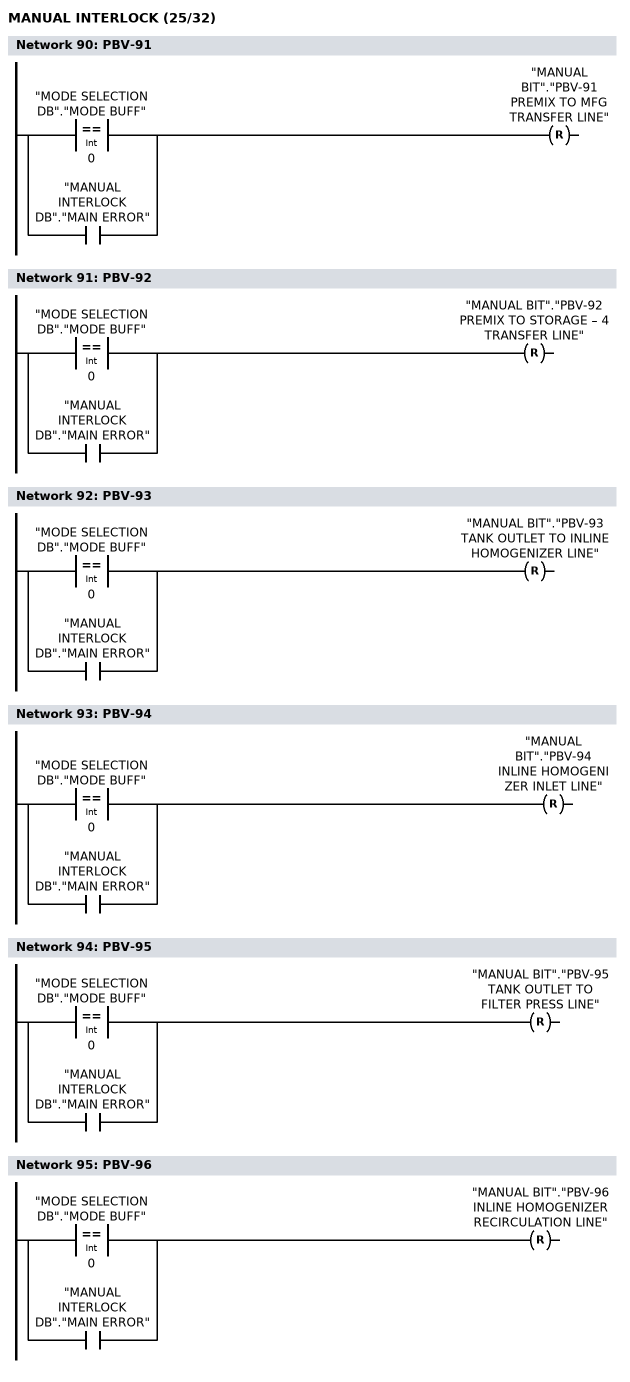
   RUNG wire#powerrail
      { S7_Templates := "SrcType := Int" } EQ_Contact(in1 := "MODE SELECTION DB"."MODE BUFF", in2 := 0)
      wire#w1
      R_Coil( "MANUAL BIT"."PBV-91 PREMIX TO MFG TRANSFER LINE" )
   END_RUNG
   RUNG wire#powerrail
      Contact( "MANUAL INTERLOCK DB"."MAIN ERROR" )
   END_RUNG wire#w1
   // the same network as SCL:
   IF ("MODE SELECTION DB"."MODE BUFF" = 0) OR "MANUAL INTERLOCK DB"."MAIN ERROR" THEN
       "MANUAL BIT"."PBV-91 PREMIX TO MFG TRANSFER LINE" := FALSE;
   END_IF;
END_REGION

REGION Network 91: PBV-92
   RUNG wire#powerrail
      { S7_Templates := "SrcType := Int" } EQ_Contact(in1 := "MODE SELECTION DB"."MODE BUFF", in2 := 0)
      wire#w1
      R_Coil( "MANUAL BIT"."PBV-92 PREMIX TO STORAGE – 4 TRANSFER LINE" )
   END_RUNG
   RUNG wire#powerrail
      Contact( "MANUAL INTERLOCK DB"."MAIN ERROR" )
   END_RUNG wire#w1
   // the same network as SCL:
   IF ("MODE SELECTION DB"."MODE BUFF" = 0) OR "MANUAL INTERLOCK DB"."MAIN ERROR" THEN
       "MANUAL BIT"."PBV-92 PREMIX TO STORAGE – 4 TRANSFER LINE" := FALSE;
   END_IF;
END_REGION

REGION Network 92: PBV-93
   RUNG wire#powerrail
      { S7_Templates := "SrcType := Int" } EQ_Contact(in1 := "MODE SELECTION DB"."MODE BUFF", in2 := 0)
      wire#w1
      R_Coil( "MANUAL BIT"."PBV-93 TANK OUTLET TO INLINE HOMOGENIZER LINE" )
   END_RUNG
   RUNG wire#powerrail
      Contact( "MANUAL INTERLOCK DB"."MAIN ERROR" )
   END_RUNG wire#w1
   // the same network as SCL:
   IF ("MODE SELECTION DB"."MODE BUFF" = 0) OR "MANUAL INTERLOCK DB"."MAIN ERROR" THEN
       "MANUAL BIT"."PBV-93 TANK OUTLET TO INLINE HOMOGENIZER LINE" := FALSE;
   END_IF;
END_REGION

REGION Network 93: PBV-94
   RUNG wire#powerrail
      { S7_Templates := "SrcType := Int" } EQ_Contact(in1 := "MODE SELECTION DB"."MODE BUFF", in2 := 0)
      wire#w1
      R_Coil( "MANUAL BIT"."PBV-94 INLINE HOMOGENIZER INLET LINE" )
   END_RUNG
   RUNG wire#powerrail
      Contact( "MANUAL INTERLOCK DB"."MAIN ERROR" )
   END_RUNG wire#w1
   // the same network as SCL:
   IF ("MODE SELECTION DB"."MODE BUFF" = 0) OR "MANUAL INTERLOCK DB"."MAIN ERROR" THEN
       "MANUAL BIT"."PBV-94 INLINE HOMOGENIZER INLET LINE" := FALSE;
   END_IF;
END_REGION

REGION Network 94: PBV-95
   RUNG wire#powerrail
      { S7_Templates := "SrcType := Int" } EQ_Contact(in1 := "MODE SELECTION DB"."MODE BUFF", in2 := 0)
      wire#w1
      R_Coil( "MANUAL BIT"."PBV-95 TANK OUTLET TO FILTER PRESS LINE" )
   END_RUNG
   RUNG wire#powerrail
      Contact( "MANUAL INTERLOCK DB"."MAIN ERROR" )
   END_RUNG wire#w1
   // the same network as SCL:
   IF ("MODE SELECTION DB"."MODE BUFF" = 0) OR "MANUAL INTERLOCK DB"."MAIN ERROR" THEN
       "MANUAL BIT"."PBV-95 TANK OUTLET TO FILTER PRESS LINE" := FALSE;
   END_IF;
END_REGION

REGION Network 95: PBV-96
   RUNG wire#powerrail
      { S7_Templates := "SrcType := Int" } EQ_Contact(in1 := "MODE SELECTION DB"."MODE BUFF", in2 := 0)
      wire#w1
      R_Coil( "MANUAL BIT"."PBV-96 INLINE HOMOGENIZER RECIRCULATION LINE" )
   END_RUNG
   RUNG wire#powerrail
      Contact( "MANUAL INTERLOCK DB"."MAIN ERROR" )
   END_RUNG wire#w1
   // the same network as SCL:
   IF ("MODE SELECTION DB"."MODE BUFF" = 0) OR "MANUAL INTERLOCK DB"."MAIN ERROR" THEN
       "MANUAL BIT"."PBV-96 INLINE HOMOGENIZER RECIRCULATION LINE" := FALSE;
   END_IF;
END_REGION

REGION Network 96: PBV-97
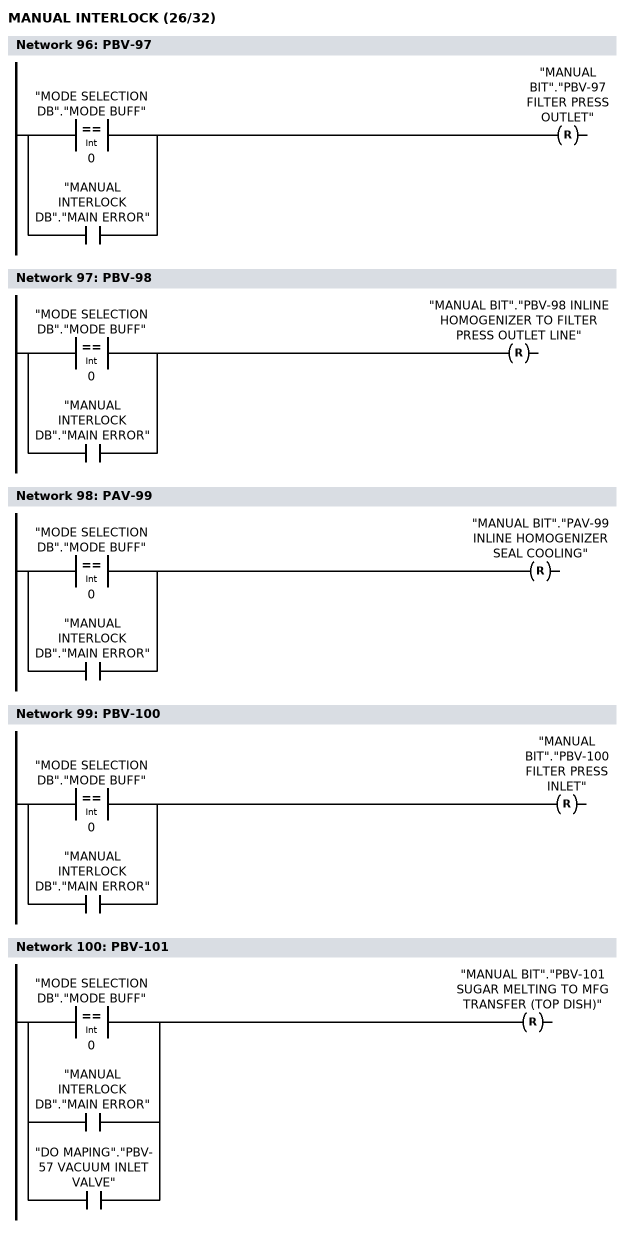
   RUNG wire#powerrail
      { S7_Templates := "SrcType := Int" } EQ_Contact(in1 := "MODE SELECTION DB"."MODE BUFF", in2 := 0)
      wire#w1
      R_Coil( "MANUAL BIT"."PBV-97 FILTER PRESS OUTLET" )
   END_RUNG
   RUNG wire#powerrail
      Contact( "MANUAL INTERLOCK DB"."MAIN ERROR" )
   END_RUNG wire#w1
   // the same network as SCL:
   IF ("MODE SELECTION DB"."MODE BUFF" = 0) OR "MANUAL INTERLOCK DB"."MAIN ERROR" THEN
       "MANUAL BIT"."PBV-97 FILTER PRESS OUTLET" := FALSE;
   END_IF;
END_REGION

REGION Network 97: PBV-98
   RUNG wire#powerrail
      { S7_Templates := "SrcType := Int" } EQ_Contact(in1 := "MODE SELECTION DB"."MODE BUFF", in2 := 0)
      wire#w1
      R_Coil( "MANUAL BIT"."PBV-98 INLINE HOMOGENIZER TO FILTER PRESS OUTLET LINE" )
   END_RUNG
   RUNG wire#powerrail
      Contact( "MANUAL INTERLOCK DB"."MAIN ERROR" )
   END_RUNG wire#w1
   // the same network as SCL:
   IF ("MODE SELECTION DB"."MODE BUFF" = 0) OR "MANUAL INTERLOCK DB"."MAIN ERROR" THEN
       "MANUAL BIT"."PBV-98 INLINE HOMOGENIZER TO FILTER PRESS OUTLET LINE" := FALSE;
   END_IF;
END_REGION

REGION Network 98: PAV-99
   RUNG wire#powerrail
      { S7_Templates := "SrcType := Int" } EQ_Contact(in1 := "MODE SELECTION DB"."MODE BUFF", in2 := 0)
      wire#w1
      R_Coil( "MANUAL BIT"."PAV-99 INLINE HOMOGENIZER SEAL COOLING" )
   END_RUNG
   RUNG wire#powerrail
      Contact( "MANUAL INTERLOCK DB"."MAIN ERROR" )
   END_RUNG wire#w1
   // the same network as SCL:
   IF ("MODE SELECTION DB"."MODE BUFF" = 0) OR "MANUAL INTERLOCK DB"."MAIN ERROR" THEN
       "MANUAL BIT"."PAV-99 INLINE HOMOGENIZER SEAL COOLING" := FALSE;
   END_IF;
END_REGION

REGION Network 99: PBV-100
   RUNG wire#powerrail
      { S7_Templates := "SrcType := Int" } EQ_Contact(in1 := "MODE SELECTION DB"."MODE BUFF", in2 := 0)
      wire#w1
      R_Coil( "MANUAL BIT"."PBV-100 FILTER PRESS INLET" )
   END_RUNG
   RUNG wire#powerrail
      Contact( "MANUAL INTERLOCK DB"."MAIN ERROR" )
   END_RUNG wire#w1
   // the same network as SCL:
   IF ("MODE SELECTION DB"."MODE BUFF" = 0) OR "MANUAL INTERLOCK DB"."MAIN ERROR" THEN
       "MANUAL BIT"."PBV-100 FILTER PRESS INLET" := FALSE;
   END_IF;
END_REGION

REGION Network 100: PBV-101
   RUNG wire#powerrail
      { S7_Templates := "SrcType := Int" } EQ_Contact(in1 := "MODE SELECTION DB"."MODE BUFF", in2 := 0)
      wire#w1
      R_Coil( "MANUAL BIT"."PBV-101 SUGAR MELTING TO MFG TRANSFER (TOP DISH)" )
   END_RUNG
   RUNG wire#powerrail
      Contact( "MANUAL INTERLOCK DB"."MAIN ERROR" )
   END_RUNG wire#w1
   RUNG wire#powerrail
      Contact( "DO MAPING"."PBV-57 VACUUM INLET VALVE" )
   END_RUNG wire#w1
   // the same network as SCL:
   IF ("MODE SELECTION DB"."MODE BUFF" = 0) OR "MANUAL INTERLOCK DB"."MAIN ERROR" OR "DO MAPING"."PBV-57 VACUUM INLET VALVE" THEN
       "MANUAL BIT"."PBV-101 SUGAR MELTING TO MFG TRANSFER (TOP DISH)" := FALSE;
   END_IF;
END_REGION

REGION Network 101: PBV-102
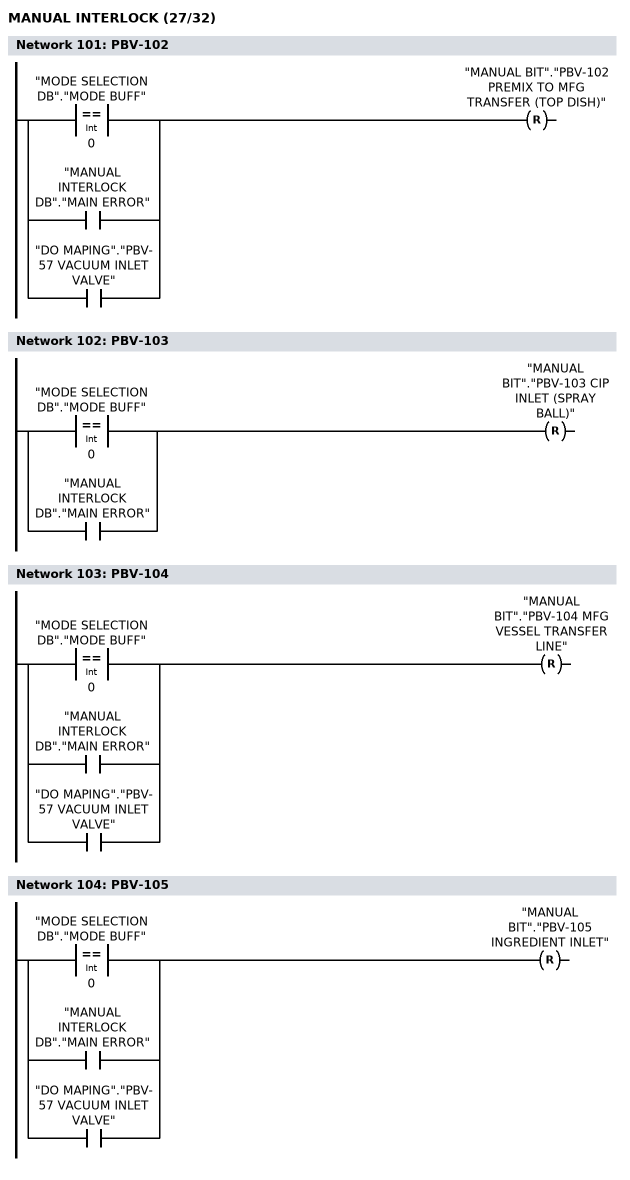
   RUNG wire#powerrail
      { S7_Templates := "SrcType := Int" } EQ_Contact(in1 := "MODE SELECTION DB"."MODE BUFF", in2 := 0)
      wire#w1
      R_Coil( "MANUAL BIT"."PBV-102 PREMIX TO MFG TRANSFER (TOP DISH)" )
   END_RUNG
   RUNG wire#powerrail
      Contact( "MANUAL INTERLOCK DB"."MAIN ERROR" )
   END_RUNG wire#w1
   RUNG wire#powerrail
      Contact( "DO MAPING"."PBV-57 VACUUM INLET VALVE" )
   END_RUNG wire#w1
   // the same network as SCL:
   IF ("MODE SELECTION DB"."MODE BUFF" = 0) OR "MANUAL INTERLOCK DB"."MAIN ERROR" OR "DO MAPING"."PBV-57 VACUUM INLET VALVE" THEN
       "MANUAL BIT"."PBV-102 PREMIX TO MFG TRANSFER (TOP DISH)" := FALSE;
   END_IF;
END_REGION

REGION Network 102: PBV-103
   RUNG wire#powerrail
      { S7_Templates := "SrcType := Int" } EQ_Contact(in1 := "MODE SELECTION DB"."MODE BUFF", in2 := 0)
      wire#w1
      R_Coil( "MANUAL BIT"."PBV-103 CIP INLET (SPRAY BALL)" )
   END_RUNG
   RUNG wire#powerrail
      Contact( "MANUAL INTERLOCK DB"."MAIN ERROR" )
   END_RUNG wire#w1
   // the same network as SCL:
   IF ("MODE SELECTION DB"."MODE BUFF" = 0) OR "MANUAL INTERLOCK DB"."MAIN ERROR" THEN
       "MANUAL BIT"."PBV-103 CIP INLET (SPRAY BALL)" := FALSE;
   END_IF;
END_REGION

REGION Network 103: PBV-104
   RUNG wire#powerrail
      { S7_Templates := "SrcType := Int" } EQ_Contact(in1 := "MODE SELECTION DB"."MODE BUFF", in2 := 0)
      wire#w1
      R_Coil( "MANUAL BIT"."PBV-104 MFG VESSEL TRANSFER LINE" )
   END_RUNG
   RUNG wire#powerrail
      Contact( "MANUAL INTERLOCK DB"."MAIN ERROR" )
   END_RUNG wire#w1
   RUNG wire#powerrail
      Contact( "DO MAPING"."PBV-57 VACUUM INLET VALVE" )
   END_RUNG wire#w1
   // the same network as SCL:
   IF ("MODE SELECTION DB"."MODE BUFF" = 0) OR "MANUAL INTERLOCK DB"."MAIN ERROR" OR "DO MAPING"."PBV-57 VACUUM INLET VALVE" THEN
       "MANUAL BIT"."PBV-104 MFG VESSEL TRANSFER LINE" := FALSE;
   END_IF;
END_REGION

REGION Network 104: PBV-105
   RUNG wire#powerrail
      { S7_Templates := "SrcType := Int" } EQ_Contact(in1 := "MODE SELECTION DB"."MODE BUFF", in2 := 0)
      wire#w1
      R_Coil( "MANUAL BIT"."PBV-105 INGREDIENT INLET" )
   END_RUNG
   RUNG wire#powerrail
      Contact( "MANUAL INTERLOCK DB"."MAIN ERROR" )
   END_RUNG wire#w1
   RUNG wire#powerrail
      Contact( "DO MAPING"."PBV-57 VACUUM INLET VALVE" )
   END_RUNG wire#w1
   // the same network as SCL:
   IF ("MODE SELECTION DB"."MODE BUFF" = 0) OR "MANUAL INTERLOCK DB"."MAIN ERROR" OR "DO MAPING"."PBV-57 VACUUM INLET VALVE" THEN
       "MANUAL BIT"."PBV-105 INGREDIENT INLET" := FALSE;
   END_IF;
END_REGION

REGION Network 105: PBV-106
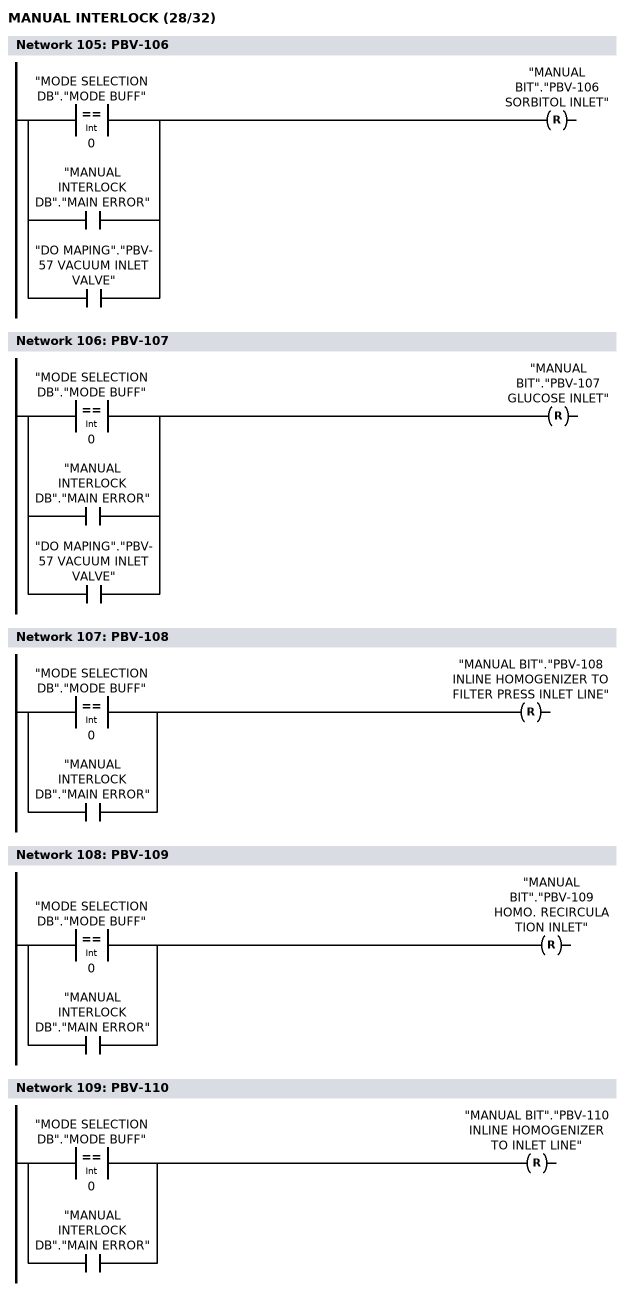
   RUNG wire#powerrail
      { S7_Templates := "SrcType := Int" } EQ_Contact(in1 := "MODE SELECTION DB"."MODE BUFF", in2 := 0)
      wire#w1
      R_Coil( "MANUAL BIT"."PBV-106 SORBITOL INLET" )
   END_RUNG
   RUNG wire#powerrail
      Contact( "MANUAL INTERLOCK DB"."MAIN ERROR" )
   END_RUNG wire#w1
   RUNG wire#powerrail
      Contact( "DO MAPING"."PBV-57 VACUUM INLET VALVE" )
   END_RUNG wire#w1
   // the same network as SCL:
   IF ("MODE SELECTION DB"."MODE BUFF" = 0) OR "MANUAL INTERLOCK DB"."MAIN ERROR" OR "DO MAPING"."PBV-57 VACUUM INLET VALVE" THEN
       "MANUAL BIT"."PBV-106 SORBITOL INLET" := FALSE;
   END_IF;
END_REGION

REGION Network 106: PBV-107
   RUNG wire#powerrail
      { S7_Templates := "SrcType := Int" } EQ_Contact(in1 := "MODE SELECTION DB"."MODE BUFF", in2 := 0)
      wire#w1
      R_Coil( "MANUAL BIT"."PBV-107 GLUCOSE INLET" )
   END_RUNG
   RUNG wire#powerrail
      Contact( "MANUAL INTERLOCK DB"."MAIN ERROR" )
   END_RUNG wire#w1
   RUNG wire#powerrail
      Contact( "DO MAPING"."PBV-57 VACUUM INLET VALVE" )
   END_RUNG wire#w1
   // the same network as SCL:
   IF ("MODE SELECTION DB"."MODE BUFF" = 0) OR "MANUAL INTERLOCK DB"."MAIN ERROR" OR "DO MAPING"."PBV-57 VACUUM INLET VALVE" THEN
       "MANUAL BIT"."PBV-107 GLUCOSE INLET" := FALSE;
   END_IF;
END_REGION

REGION Network 107: PBV-108
   RUNG wire#powerrail
      { S7_Templates := "SrcType := Int" } EQ_Contact(in1 := "MODE SELECTION DB"."MODE BUFF", in2 := 0)
      wire#w1
      R_Coil( "MANUAL BIT"."PBV-108 INLINE HOMOGENIZER TO FILTER PRESS INLET LINE" )
   END_RUNG
   RUNG wire#powerrail
      Contact( "MANUAL INTERLOCK DB"."MAIN ERROR" )
   END_RUNG wire#w1
   // the same network as SCL:
   IF ("MODE SELECTION DB"."MODE BUFF" = 0) OR "MANUAL INTERLOCK DB"."MAIN ERROR" THEN
       "MANUAL BIT"."PBV-108 INLINE HOMOGENIZER TO FILTER PRESS INLET LINE" := FALSE;
   END_IF;
END_REGION

REGION Network 108: PBV-109
   RUNG wire#powerrail
      { S7_Templates := "SrcType := Int" } EQ_Contact(in1 := "MODE SELECTION DB"."MODE BUFF", in2 := 0)
      wire#w1
      R_Coil( "MANUAL BIT"."PBV-109 HOMO. RECIRCULATION INLET" )
   END_RUNG
   RUNG wire#powerrail
      Contact( "MANUAL INTERLOCK DB"."MAIN ERROR" )
   END_RUNG wire#w1
   // the same network as SCL:
   IF ("MODE SELECTION DB"."MODE BUFF" = 0) OR "MANUAL INTERLOCK DB"."MAIN ERROR" THEN
       "MANUAL BIT"."PBV-109 HOMO. RECIRCULATION INLET" := FALSE;
   END_IF;
END_REGION

REGION Network 109: PBV-110
   RUNG wire#powerrail
      { S7_Templates := "SrcType := Int" } EQ_Contact(in1 := "MODE SELECTION DB"."MODE BUFF", in2 := 0)
      wire#w1
      R_Coil( "MANUAL BIT"."PBV-110 INLINE HOMOGENIZER TO INLET LINE" )
   END_RUNG
   RUNG wire#powerrail
      Contact( "MANUAL INTERLOCK DB"."MAIN ERROR" )
   END_RUNG wire#w1
   // the same network as SCL:
   IF ("MODE SELECTION DB"."MODE BUFF" = 0) OR "MANUAL INTERLOCK DB"."MAIN ERROR" THEN
       "MANUAL BIT"."PBV-110 INLINE HOMOGENIZER TO INLET LINE" := FALSE;
   END_IF;
END_REGION

REGION Network 110: PBV-111
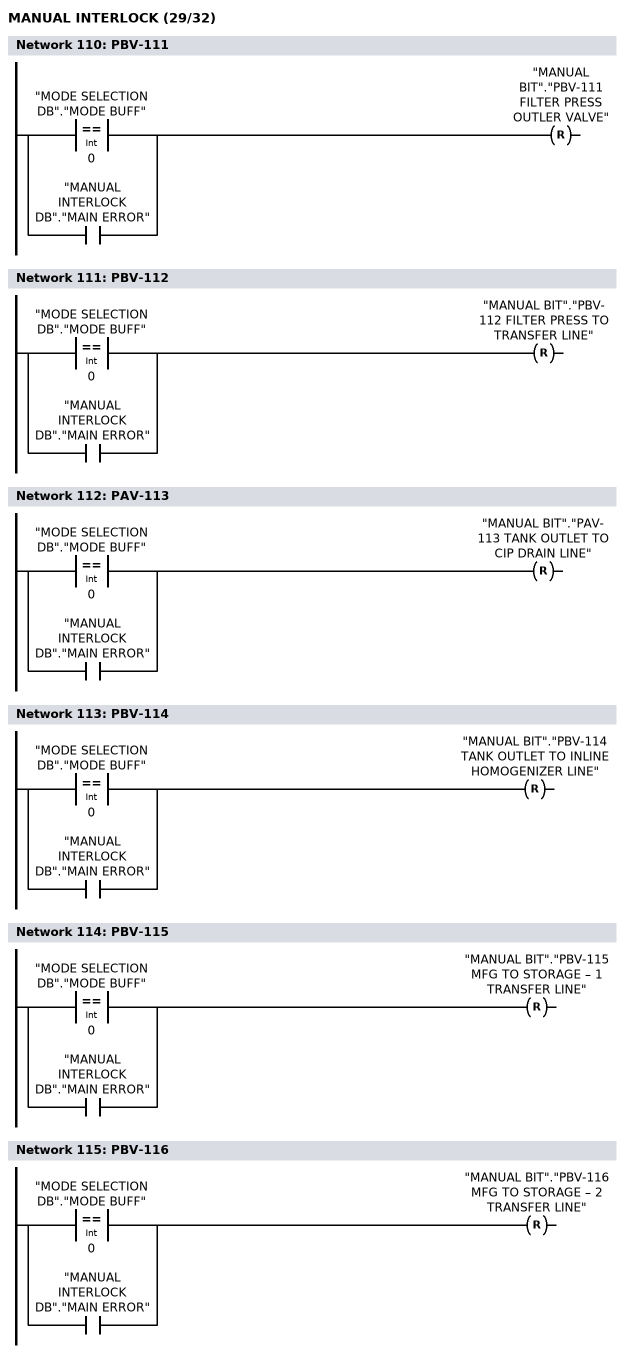
   RUNG wire#powerrail
      { S7_Templates := "SrcType := Int" } EQ_Contact(in1 := "MODE SELECTION DB"."MODE BUFF", in2 := 0)
      wire#w1
      R_Coil( "MANUAL BIT"."PBV-111 FILTER PRESS OUTLER VALVE" )
   END_RUNG
   RUNG wire#powerrail
      Contact( "MANUAL INTERLOCK DB"."MAIN ERROR" )
   END_RUNG wire#w1
   // the same network as SCL:
   IF ("MODE SELECTION DB"."MODE BUFF" = 0) OR "MANUAL INTERLOCK DB"."MAIN ERROR" THEN
       "MANUAL BIT"."PBV-111 FILTER PRESS OUTLER VALVE" := FALSE;
   END_IF;
END_REGION

REGION Network 111: PBV-112
   RUNG wire#powerrail
      { S7_Templates := "SrcType := Int" } EQ_Contact(in1 := "MODE SELECTION DB"."MODE BUFF", in2 := 0)
      wire#w1
      R_Coil( "MANUAL BIT"."PBV-112 FILTER PRESS TO TRANSFER LINE" )
   END_RUNG
   RUNG wire#powerrail
      Contact( "MANUAL INTERLOCK DB"."MAIN ERROR" )
   END_RUNG wire#w1
   // the same network as SCL:
   IF ("MODE SELECTION DB"."MODE BUFF" = 0) OR "MANUAL INTERLOCK DB"."MAIN ERROR" THEN
       "MANUAL BIT"."PBV-112 FILTER PRESS TO TRANSFER LINE" := FALSE;
   END_IF;
END_REGION

REGION Network 112: PAV-113
   RUNG wire#powerrail
      { S7_Templates := "SrcType := Int" } EQ_Contact(in1 := "MODE SELECTION DB"."MODE BUFF", in2 := 0)
      wire#w1
      R_Coil( "MANUAL BIT"."PAV-113 TANK OUTLET TO CIP DRAIN LINE" )
   END_RUNG
   RUNG wire#powerrail
      Contact( "MANUAL INTERLOCK DB"."MAIN ERROR" )
   END_RUNG wire#w1
   // the same network as SCL:
   IF ("MODE SELECTION DB"."MODE BUFF" = 0) OR "MANUAL INTERLOCK DB"."MAIN ERROR" THEN
       "MANUAL BIT"."PAV-113 TANK OUTLET TO CIP DRAIN LINE" := FALSE;
   END_IF;
END_REGION

REGION Network 113: PBV-114
   RUNG wire#powerrail
      { S7_Templates := "SrcType := Int" } EQ_Contact(in1 := "MODE SELECTION DB"."MODE BUFF", in2 := 0)
      wire#w1
      R_Coil( "MANUAL BIT"."PBV-114 TANK OUTLET TO INLINE HOMOGENIZER LINE" )
   END_RUNG
   RUNG wire#powerrail
      Contact( "MANUAL INTERLOCK DB"."MAIN ERROR" )
   END_RUNG wire#w1
   // the same network as SCL:
   IF ("MODE SELECTION DB"."MODE BUFF" = 0) OR "MANUAL INTERLOCK DB"."MAIN ERROR" THEN
       "MANUAL BIT"."PBV-114 TANK OUTLET TO INLINE HOMOGENIZER LINE" := FALSE;
   END_IF;
END_REGION

REGION Network 114: PBV-115
   RUNG wire#powerrail
      { S7_Templates := "SrcType := Int" } EQ_Contact(in1 := "MODE SELECTION DB"."MODE BUFF", in2 := 0)
      wire#w1
      R_Coil( "MANUAL BIT"."PBV-115 MFG TO STORAGE – 1 TRANSFER LINE" )
   END_RUNG
   RUNG wire#powerrail
      Contact( "MANUAL INTERLOCK DB"."MAIN ERROR" )
   END_RUNG wire#w1
   // the same network as SCL:
   IF ("MODE SELECTION DB"."MODE BUFF" = 0) OR "MANUAL INTERLOCK DB"."MAIN ERROR" THEN
       "MANUAL BIT"."PBV-115 MFG TO STORAGE – 1 TRANSFER LINE" := FALSE;
   END_IF;
END_REGION

REGION Network 115: PBV-116
   RUNG wire#powerrail
      { S7_Templates := "SrcType := Int" } EQ_Contact(in1 := "MODE SELECTION DB"."MODE BUFF", in2 := 0)
      wire#w1
      R_Coil( "MANUAL BIT"."PBV-116 MFG TO STORAGE – 2 TRANSFER LINE" )
   END_RUNG
   RUNG wire#powerrail
      Contact( "MANUAL INTERLOCK DB"."MAIN ERROR" )
   END_RUNG wire#w1
   // the same network as SCL:
   IF ("MODE SELECTION DB"."MODE BUFF" = 0) OR "MANUAL INTERLOCK DB"."MAIN ERROR" THEN
       "MANUAL BIT"."PBV-116 MFG TO STORAGE – 2 TRANSFER LINE" := FALSE;
   END_IF;
END_REGION

REGION Network 116: PBV-117
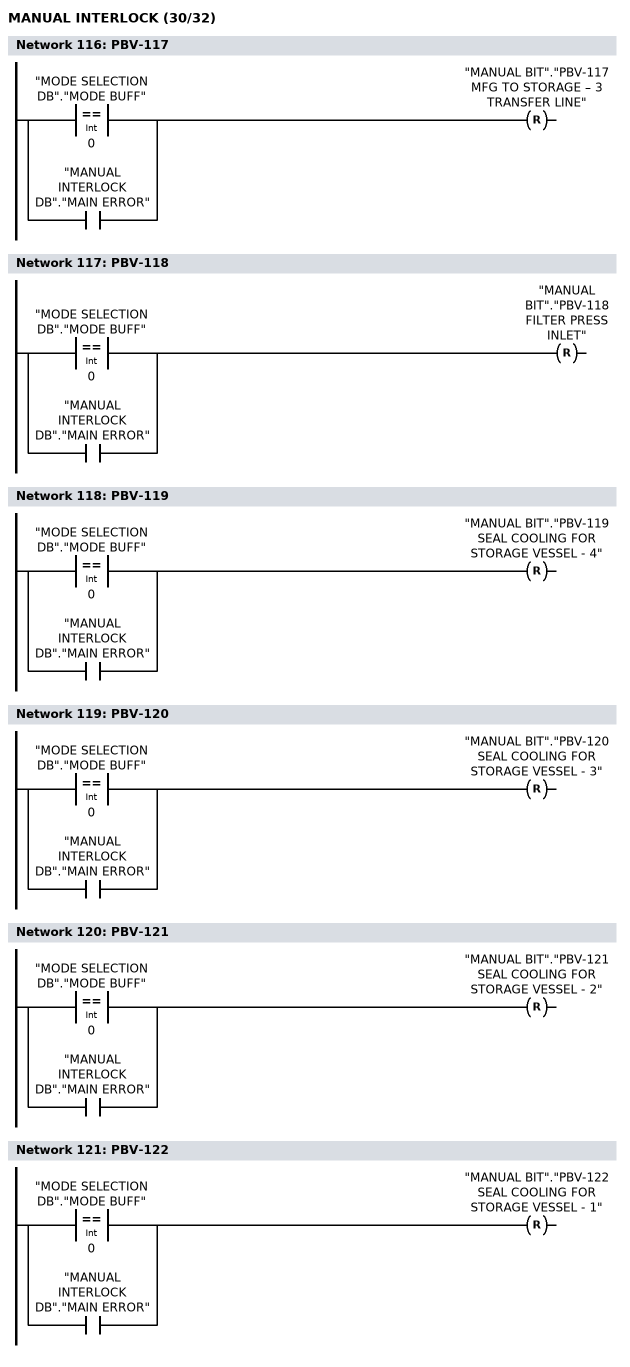
   RUNG wire#powerrail
      { S7_Templates := "SrcType := Int" } EQ_Contact(in1 := "MODE SELECTION DB"."MODE BUFF", in2 := 0)
      wire#w1
      R_Coil( "MANUAL BIT"."PBV-117 MFG TO STORAGE – 3 TRANSFER LINE" )
   END_RUNG
   RUNG wire#powerrail
      Contact( "MANUAL INTERLOCK DB"."MAIN ERROR" )
   END_RUNG wire#w1
   // the same network as SCL:
   IF ("MODE SELECTION DB"."MODE BUFF" = 0) OR "MANUAL INTERLOCK DB"."MAIN ERROR" THEN
       "MANUAL BIT"."PBV-117 MFG TO STORAGE – 3 TRANSFER LINE" := FALSE;
   END_IF;
END_REGION

REGION Network 117: PBV-118
   RUNG wire#powerrail
      { S7_Templates := "SrcType := Int" } EQ_Contact(in1 := "MODE SELECTION DB"."MODE BUFF", in2 := 0)
      wire#w1
      R_Coil( "MANUAL BIT"."PBV-118 FILTER PRESS INLET" )
   END_RUNG
   RUNG wire#powerrail
      Contact( "MANUAL INTERLOCK DB"."MAIN ERROR" )
   END_RUNG wire#w1
   // the same network as SCL:
   IF ("MODE SELECTION DB"."MODE BUFF" = 0) OR "MANUAL INTERLOCK DB"."MAIN ERROR" THEN
       "MANUAL BIT"."PBV-118 FILTER PRESS INLET" := FALSE;
   END_IF;
END_REGION

REGION Network 118: PBV-119
   RUNG wire#powerrail
      { S7_Templates := "SrcType := Int" } EQ_Contact(in1 := "MODE SELECTION DB"."MODE BUFF", in2 := 0)
      wire#w1
      R_Coil( "MANUAL BIT"."PBV-119 SEAL COOLING FOR STORAGE VESSEL - 4" )
   END_RUNG
   RUNG wire#powerrail
      Contact( "MANUAL INTERLOCK DB"."MAIN ERROR" )
   END_RUNG wire#w1
   // the same network as SCL:
   IF ("MODE SELECTION DB"."MODE BUFF" = 0) OR "MANUAL INTERLOCK DB"."MAIN ERROR" THEN
       "MANUAL BIT"."PBV-119 SEAL COOLING FOR STORAGE VESSEL - 4" := FALSE;
   END_IF;
END_REGION

REGION Network 119: PBV-120
   RUNG wire#powerrail
      { S7_Templates := "SrcType := Int" } EQ_Contact(in1 := "MODE SELECTION DB"."MODE BUFF", in2 := 0)
      wire#w1
      R_Coil( "MANUAL BIT"."PBV-120 SEAL COOLING FOR STORAGE VESSEL - 3" )
   END_RUNG
   RUNG wire#powerrail
      Contact( "MANUAL INTERLOCK DB"."MAIN ERROR" )
   END_RUNG wire#w1
   // the same network as SCL:
   IF ("MODE SELECTION DB"."MODE BUFF" = 0) OR "MANUAL INTERLOCK DB"."MAIN ERROR" THEN
       "MANUAL BIT"."PBV-120 SEAL COOLING FOR STORAGE VESSEL - 3" := FALSE;
   END_IF;
END_REGION

REGION Network 120: PBV-121
   RUNG wire#powerrail
      { S7_Templates := "SrcType := Int" } EQ_Contact(in1 := "MODE SELECTION DB"."MODE BUFF", in2 := 0)
      wire#w1
      R_Coil( "MANUAL BIT"."PBV-121 SEAL COOLING FOR STORAGE VESSEL - 2" )
   END_RUNG
   RUNG wire#powerrail
      Contact( "MANUAL INTERLOCK DB"."MAIN ERROR" )
   END_RUNG wire#w1
   // the same network as SCL:
   IF ("MODE SELECTION DB"."MODE BUFF" = 0) OR "MANUAL INTERLOCK DB"."MAIN ERROR" THEN
       "MANUAL BIT"."PBV-121 SEAL COOLING FOR STORAGE VESSEL - 2" := FALSE;
   END_IF;
END_REGION

REGION Network 121: PBV-122
   RUNG wire#powerrail
      { S7_Templates := "SrcType := Int" } EQ_Contact(in1 := "MODE SELECTION DB"."MODE BUFF", in2 := 0)
      wire#w1
      R_Coil( "MANUAL BIT"."PBV-122 SEAL COOLING FOR STORAGE VESSEL - 1" )
   END_RUNG
   RUNG wire#powerrail
      Contact( "MANUAL INTERLOCK DB"."MAIN ERROR" )
   END_RUNG wire#w1
   // the same network as SCL:
   IF ("MODE SELECTION DB"."MODE BUFF" = 0) OR "MANUAL INTERLOCK DB"."MAIN ERROR" THEN
       "MANUAL BIT"."PBV-122 SEAL COOLING FOR STORAGE VESSEL - 1" := FALSE;
   END_IF;
END_REGION

REGION Network 122: PBV-123
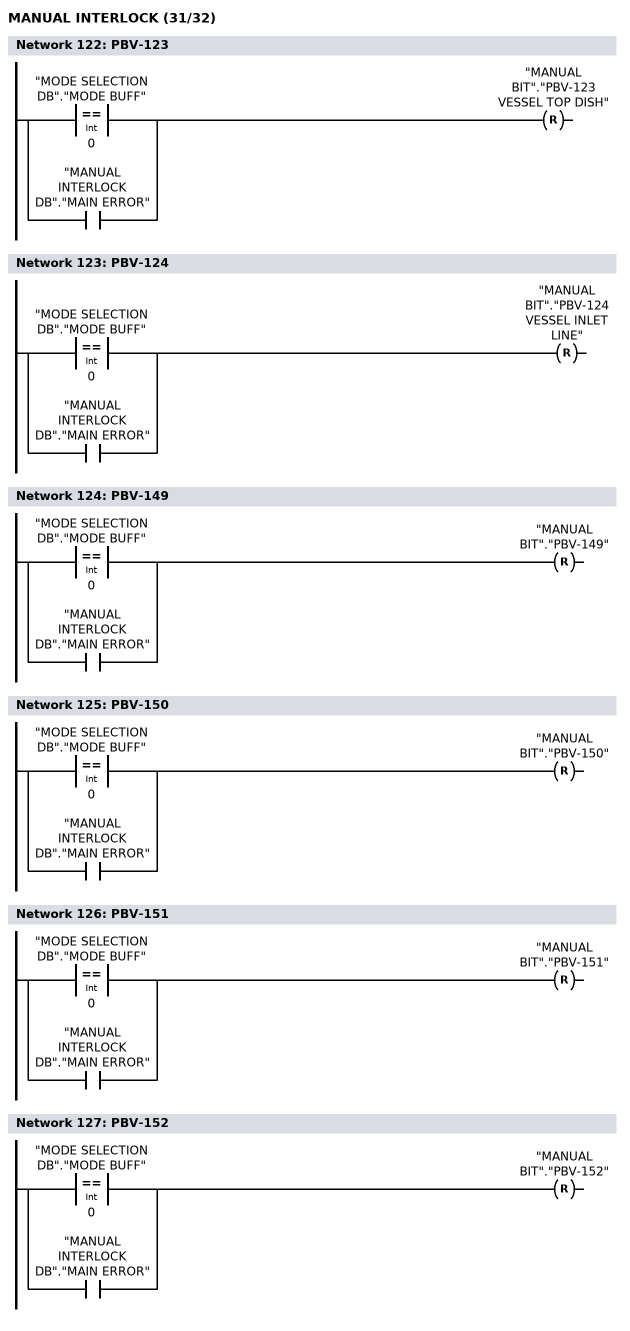
   RUNG wire#powerrail
      { S7_Templates := "SrcType := Int" } EQ_Contact(in1 := "MODE SELECTION DB"."MODE BUFF", in2 := 0)
      wire#w1
      R_Coil( "MANUAL BIT"."PBV-123 VESSEL TOP DISH" )
   END_RUNG
   RUNG wire#powerrail
      Contact( "MANUAL INTERLOCK DB"."MAIN ERROR" )
   END_RUNG wire#w1
   // the same network as SCL:
   IF ("MODE SELECTION DB"."MODE BUFF" = 0) OR "MANUAL INTERLOCK DB"."MAIN ERROR" THEN
       "MANUAL BIT"."PBV-123 VESSEL TOP DISH" := FALSE;
   END_IF;
END_REGION

REGION Network 123: PBV-124
   RUNG wire#powerrail
      { S7_Templates := "SrcType := Int" } EQ_Contact(in1 := "MODE SELECTION DB"."MODE BUFF", in2 := 0)
      wire#w1
      R_Coil( "MANUAL BIT"."PBV-124 VESSEL INLET LINE" )
   END_RUNG
   RUNG wire#powerrail
      Contact( "MANUAL INTERLOCK DB"."MAIN ERROR" )
   END_RUNG wire#w1
   // the same network as SCL:
   IF ("MODE SELECTION DB"."MODE BUFF" = 0) OR "MANUAL INTERLOCK DB"."MAIN ERROR" THEN
       "MANUAL BIT"."PBV-124 VESSEL INLET LINE" := FALSE;
   END_IF;
END_REGION

REGION Network 124: PBV-149
   RUNG wire#powerrail
      { S7_Templates := "SrcType := Int" } EQ_Contact(in1 := "MODE SELECTION DB"."MODE BUFF", in2 := 0)
      wire#w1
      R_Coil( "MANUAL BIT"."PBV-149" )
   END_RUNG
   RUNG wire#powerrail
      Contact( "MANUAL INTERLOCK DB"."MAIN ERROR" )
   END_RUNG wire#w1
   // the same network as SCL:
   IF ("MODE SELECTION DB"."MODE BUFF" = 0) OR "MANUAL INTERLOCK DB"."MAIN ERROR" THEN
       "MANUAL BIT"."PBV-149" := FALSE;
   END_IF;
END_REGION

REGION Network 125: PBV-150
   RUNG wire#powerrail
      { S7_Templates := "SrcType := Int" } EQ_Contact(in1 := "MODE SELECTION DB"."MODE BUFF", in2 := 0)
      wire#w1
      R_Coil( "MANUAL BIT"."PBV-150" )
   END_RUNG
   RUNG wire#powerrail
      Contact( "MANUAL INTERLOCK DB"."MAIN ERROR" )
   END_RUNG wire#w1
   // the same network as SCL:
   IF ("MODE SELECTION DB"."MODE BUFF" = 0) OR "MANUAL INTERLOCK DB"."MAIN ERROR" THEN
       "MANUAL BIT"."PBV-150" := FALSE;
   END_IF;
END_REGION

REGION Network 126: PBV-151
   RUNG wire#powerrail
      { S7_Templates := "SrcType := Int" } EQ_Contact(in1 := "MODE SELECTION DB"."MODE BUFF", in2 := 0)
      wire#w1
      R_Coil( "MANUAL BIT"."PBV-151" )
   END_RUNG
   RUNG wire#powerrail
      Contact( "MANUAL INTERLOCK DB"."MAIN ERROR" )
   END_RUNG wire#w1
   // the same network as SCL:
   IF ("MODE SELECTION DB"."MODE BUFF" = 0) OR "MANUAL INTERLOCK DB"."MAIN ERROR" THEN
       "MANUAL BIT"."PBV-151" := FALSE;
   END_IF;
END_REGION

REGION Network 127: PBV-152
   RUNG wire#powerrail
      { S7_Templates := "SrcType := Int" } EQ_Contact(in1 := "MODE SELECTION DB"."MODE BUFF", in2 := 0)
      wire#w1
      R_Coil( "MANUAL BIT"."PBV-152" )
   END_RUNG
   RUNG wire#powerrail
      Contact( "MANUAL INTERLOCK DB"."MAIN ERROR" )
   END_RUNG wire#w1
   // the same network as SCL:
   IF ("MODE SELECTION DB"."MODE BUFF" = 0) OR "MANUAL INTERLOCK DB"."MAIN ERROR" THEN
       "MANUAL BIT"."PBV-152" := FALSE;
   END_IF;
END_REGION

REGION Network 128: PBV-153
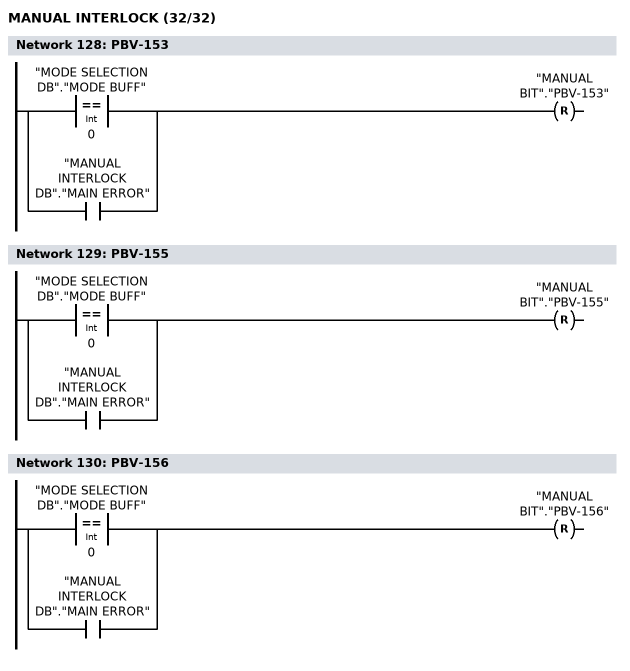
   RUNG wire#powerrail
      { S7_Templates := "SrcType := Int" } EQ_Contact(in1 := "MODE SELECTION DB"."MODE BUFF", in2 := 0)
      wire#w1
      R_Coil( "MANUAL BIT"."PBV-153" )
   END_RUNG
   RUNG wire#powerrail
      Contact( "MANUAL INTERLOCK DB"."MAIN ERROR" )
   END_RUNG wire#w1
   // the same network as SCL:
   IF ("MODE SELECTION DB"."MODE BUFF" = 0) OR "MANUAL INTERLOCK DB"."MAIN ERROR" THEN
       "MANUAL BIT"."PBV-153" := FALSE;
   END_IF;
END_REGION

REGION Network 129: PBV-155
   RUNG wire#powerrail
      { S7_Templates := "SrcType := Int" } EQ_Contact(in1 := "MODE SELECTION DB"."MODE BUFF", in2 := 0)
      wire#w1
      R_Coil( "MANUAL BIT"."PBV-155" )
   END_RUNG
   RUNG wire#powerrail
      Contact( "MANUAL INTERLOCK DB"."MAIN ERROR" )
   END_RUNG wire#w1
   // the same network as SCL:
   IF ("MODE SELECTION DB"."MODE BUFF" = 0) OR "MANUAL INTERLOCK DB"."MAIN ERROR" THEN
       "MANUAL BIT"."PBV-155" := FALSE;
   END_IF;
END_REGION

REGION Network 130: PBV-156
   RUNG wire#powerrail
      { S7_Templates := "SrcType := Int" } EQ_Contact(in1 := "MODE SELECTION DB"."MODE BUFF", in2 := 0)
      wire#w1
      R_Coil( "MANUAL BIT"."PBV-156" )
   END_RUNG
   RUNG wire#powerrail
      Contact( "MANUAL INTERLOCK DB"."MAIN ERROR" )
   END_RUNG wire#w1
   // the same network as SCL:
   IF ("MODE SELECTION DB"."MODE BUFF" = 0) OR "MANUAL INTERLOCK DB"."MAIN ERROR" THEN
       "MANUAL BIT"."PBV-156" := FALSE;
   END_IF;
END_REGION
END_FUNCTION
